PROGRAM task1
VAr
END_VAR

END_PROGRAM

(* stored: Version 1.1.0.1, ProductVersion 3.1.4024.15
   POU task1: Id {20a40416-a3f2-4129-a137-0b4baf41b1bb}, SpecialFunc None *)
